FUNCTION AdditionFunction : REAL
VAR_INPUT
	i_rValueA : REAL;
	i_rValueB : REAL;
END_VAR
VAR
END_VAR

AdditionFunction := i_rValueA + i_rValueB;

END_FUNCTION

(* stored: Version 1.1.0.1, ProductVersion 3.1.4022.12
   POU AdditionFunction: Id {5777d249-9682-4539-ac0b-1f1699f5cd39}, SpecialFunc None *)
